TYPE DUT_IO_Valve :
STRUCT
	I_isOpen AT %I* : BOOL := FALSE;
	I_isClosed AT %I*   : BOOL := FALSE;
	I_isHealthy AT %I* : BOOL := FALSE;
	O_setOpen AT %Q*   : BOOL := FALSE;
END_STRUCT
END_TYPE

(* stored: Version 1.1.0.1, ProductVersion 3.1.4024.12
   DUT DUT_IO_Valve: Id {4268dc97-dd5f-4104-9a13-78dc9484310a} *)
